// Device/Application/可视化/TlCtrl
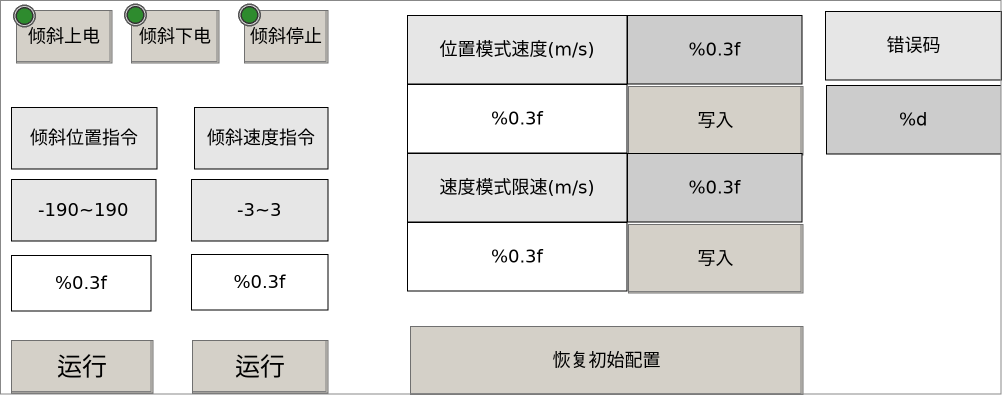
VISUALIZATION TlCtrl  // 1002x395
    Button (131,10 88x53), "倾斜下电"
        OnMouseClick: execute { GVL.Axis3Local.iMode:=0; }
    Button (16,10 96x53), "倾斜上电"
        OnMouseClick: execute { GVL.Axis3Local.iMode:=1; }
    Lamp1 (6,3 37x26), variable: GVL.Axis3Status.bServo_Enable, style: Lamp-Lamp1-Green
    Lamp1 (117,2 37x26), variable: NOT(GVL.Axis3Status.bServo_Enable), style: Lamp-Lamp1-Green
    Button (244,10 84x53), "倾斜停止"
        OnMouseClick: execute { GVL.Axis3Local.iMode:=7; }
    Lamp1 (231,2 37x26), variable: NOT(GVL.Axis3Status.Moving), style: Lamp-Lamp1-Green
    Rectangle (11,107 146x62), "倾斜位置指令"
    Rectangle (11,255 140x56), "%0.3f", text variable: TiV.rPosCmd
        OnMouseClick: write the text variable via Default, min -190, max 190
    Button (11,340 142x53), "运行"
        OnMouseClick: execute {
            GVL.Axis3Local.rPosCmd:=-GVL.TiV.rPosCmd;
            GVL.Axis3Local.iMode:=4;
            GVL.Axis3Local.bPIDEnable:=TRUE;
        }
    Rectangle (194,107 134x62), "倾斜速度指令"
    Rectangle (191,254 137x56), "%0.3f", text variable: TiV.rVelCmd
        OnMouseClick: write the text variable via Default, min -11, max 11
    Button (192,340 136x53), "运行"
        OnMouseClick: execute { GVL.Axis3Local.rVelCmd:=GVL.TiV.rVelCmd*(-1); GVL.Axis3Local.iMode:=3; }
    Rectangle (11,179 145x62), "-190~190"
    Rectangle (191,179 137x62), "-3~3"
    Rectangle (627,15 175x69), "%0.3f", text variable: Axis3Local.Pos_Vel
    Rectangle (407,15 220x69), "位置模式速度(m/s)"
    Rectangle (407,84 220x69), "%0.3f", text variable: TiV.Pos_Vel
        OnMouseClick: write the text variable via Edit, min -15.5, max 15.5
    Button (628,86 175x69), "写入"
        OnMouseClick: execute { Axis3Local.Pos_Vel:=TiV.Pos_Vel; }
    Rectangle (627,153 175x69), "%0.3f", text variable: Axis3Local.rVel_Limit
    Rectangle (407,153 220x69), "速度模式限速(m/s)"
    Rectangle (407,222 220x69), "%0.3f", text variable: TiV.rVel_Limit
        OnMouseClick: write the text variable via Edit, min -15.5, max 15.5
    Button (628,224 175x69), "写入"
        OnMouseClick: execute { Axis3Local.rVel_Limit:=TiV.rVel_Limit; }
    Button (410,326 393x69), "恢复初始配置"
        OnMouseClick: execute { Axis3Local.rVel_Limit:=3; Axis3Local.Pos_Vel:=4; }
    Rectangle (826,85 175x69), "%d", text variable: GVL.eTiErrorcode
    Rectangle (825,11 177x69), "错误码"
END_VISUALIZATION

// Device/Application/可视化/north
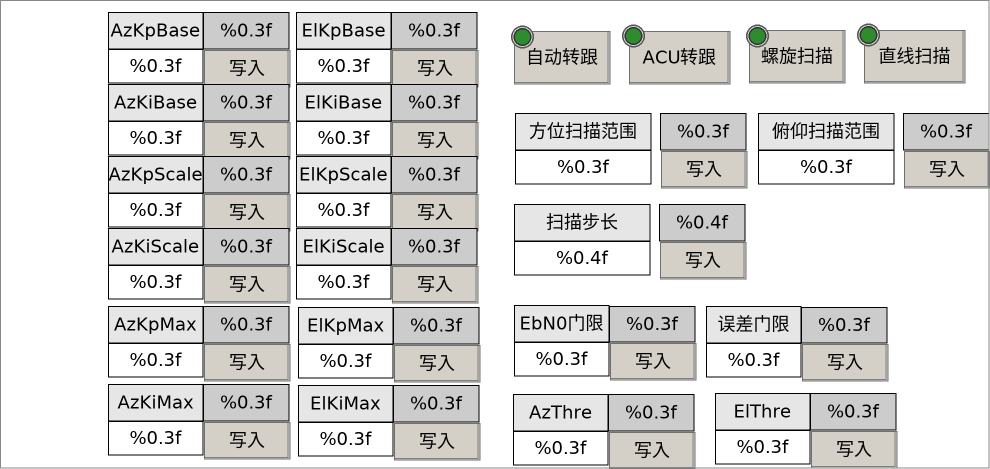
VISUALIZATION north  // 990x469
    Rectangle (203,12 86x37), "%0.3f", text variable: PersistentVars.rAzKpBase
    Rectangle (108,12 95x37), "AzKpBase"
    Rectangle (108,49 95x34), "%0.3f", text variable: GVL.rvAzKpBase
        OnMouseClick: write the text variable via Edit, min -100, max 100
    Button (204,50 86x37), "写入"
        OnMouseClick: execute { persistentvars.rAzKpBase := gvl.rvAzKpBase; }
    Rectangle (203,84 86x37), "%0.3f", text variable: PersistentVars.rAzKiBase
    Button (204,122 86x37), "写入"
        OnMouseClick: execute { persistentvars.rAzKiBase := gvl.rvAzKiBase; }
    Rectangle (203,156 86x37), "%0.3f", text variable: PersistentVars.rAzKpscale
    Button (204,194 86x37), "写入"
        OnMouseClick: execute { persistentvars.rAzKpScale := gvl.rvAzKpScale; }
    Rectangle (203,228 86x37), "%0.3f", text variable: PersistentVars.rAzKiscale
    Button (204,266 86x37), "写入"
        OnMouseClick: execute { persistentvars.rAzKiScale := gvl.rvAzKiScale; }
    Rectangle (108,84 95x37), "AzKiBase"
    Rectangle (108,121 95x34), "%0.3f", text variable: GVL.rvAzKiBase
        OnMouseClick: write the text variable via Edit, min -100, max 100
    Rectangle (108,156 95x37), "AzKpScale"
    Rectangle (108,193 95x34), "%0.3f", text variable: GVL.rvAzKpscale
        OnMouseClick: write the text variable via Edit, min -100, max 100
    Rectangle (108,228 95x37), "AzKiScale"
    Rectangle (108,265 95x34), "%0.3f", text variable: GVL.rvAzKiscale
        OnMouseClick: write the text variable via Edit, min -100, max 100
    Rectangle (391,12 86x37), "%0.3f", text variable: PersistentVars.rElKpBase
    Rectangle (296,12 95x37), "ElKpBase"
    Rectangle (296,49 95x34), "%0.3f", text variable: GVL.rvElKpBase
        OnMouseClick: write the text variable via Edit, min -100, max 100
    Button (392,50 86x37), "写入"
        OnMouseClick: execute { persistentvars.rElKpBase := gvl.rvElKpBase; }
    Rectangle (391,84 86x37), "%0.3f", text variable: PersistentVars.rElKiBase
    Button (392,122 86x37), "写入"
        OnMouseClick: execute { persistentvars.rElKiBase := gvl.rvElKiBase; }
    Rectangle (391,156 86x37), "%0.3f", text variable: PersistentVars.rElKpscale
    Button (392,194 86x37), "写入"
        OnMouseClick: execute { persistentvars.rElKpScale := gvl.rvElKpScale; }
    Rectangle (391,228 86x37), "%0.3f", text variable: PersistentVars.rElKiscale
    Button (392,266 86x37), "写入"
        OnMouseClick: execute { persistentvars.rElKiScale := gvl.rvElKiScale; }
    Rectangle (296,84 95x37), "ElKiBase"
    Rectangle (296,121 95x34), "%0.3f", text variable: GVL.rvElKiBase
        OnMouseClick: write the text variable via Edit, min -100, max 100
    Rectangle (296,156 95x37), "ElKpScale"
    Rectangle (296,193 95x34), "%0.3f", text variable: GVL.rvElKpscale
        OnMouseClick: write the text variable via Edit, min -100, max 100
    Rectangle (296,228 95x37), "ElKiScale"
    Rectangle (296,265 95x34), "%0.3f", text variable: GVL.rvElKiscale
        OnMouseClick: write the text variable via Edit, min -100, max 100
    Rectangle (203,306 86x37), "%0.3f", text variable: PersistentVars.rAzKpMax
    Rectangle (108,306 95x37), "AzKpMax"
    Rectangle (108,343 95x34), "%0.3f", text variable: GVL.rvAzKpMax
        OnMouseClick: write the text variable via Edit, min -100, max 100
    Button (204,344 86x37), "写入"
        OnMouseClick: execute { persistentvars.rAzKpMax := gvl.rvAzKpMax; }
    Rectangle (203,384 86x37), "%0.3f", text variable: PersistentVars.rAzKiMax
    Rectangle (108,384 95x37), "AzKiMax"
    Rectangle (108,421 95x34), "%0.3f", text variable: GVL.rvAzKiMax
        OnMouseClick: write the text variable via Edit, min -100, max 100
    Button (204,422 86x37), "写入"
        OnMouseClick: execute { persistentvars.rAzKiMax := gvl.rvAzKiMax; }
    Rectangle (393,307 86x37), "%0.3f", text variable: PersistentVars.rElKpMax
    Rectangle (298,307 95x37), "ElKpMax"
    Rectangle (298,344 95x34), "%0.3f", text variable: GVL.rvElKpMax
        OnMouseClick: write the text variable via Edit, min -100, max 100
    Button (394,345 86x37), "写入"
        OnMouseClick: execute { persistentvars.rElKpMax := gvl.rvElKpMax; }
    Rectangle (393,385 86x37), "%0.3f", text variable: PersistentVars.rElKiMax
    Rectangle (298,385 95x37), "ElKiMax"
    Rectangle (298,422 95x34), "%0.3f", text variable: GVL.rvElKiMax
        OnMouseClick: write the text variable via Edit, min -100, max 100
    Button (394,423 86x37), "写入"
        OnMouseClick: execute { persistentvars.rElKiMax := gvl.rvElKiMax; }
    Rectangle (608,394 86x37), "%0.3f", text variable: PersistentVars.rAzThre
    Rectangle (513,394 95x37), "AzThre"
    Rectangle (513,431 95x34), "%0.3f", text variable: GVL.rvAzThre
        OnMouseClick: write the text variable via Edit, min -100, max 100
    Button (609,432 86x37), "写入"
        OnMouseClick: execute { persistentvars.rAzThre := gvl.rvAzThre; }
    Rectangle (810,393 86x37), "%0.3f", text variable: PersistentVars.rElThre
    Rectangle (715,393 95x37), "ElThre"
    Rectangle (715,430 95x34), "%0.3f", text variable: GVL.rvElThre
        OnMouseClick: write the text variable via Edit, min -100, max 100
    Button (811,431 86x37), "写入"
        OnMouseClick: execute { persistentvars.rElThre := gvl.rvElThre; }
    Rectangle (609,306 86x36), "%0.3f", text variable: PersistentVars.rEbN0LockThre
    Rectangle (514,305 95x37), "EbN0门限"
    Rectangle (514,342 95x34), "%0.3f", text variable: GVL.rEbN0LockThreEdit
        OnMouseClick: write the text variable via Edit, min 0, max 30
    Button (610,343 86x37), "写入"
        OnMouseClick: execute { PersistentVars.rEbN0LockThre := GVL.rEbN0LockThreEdit; }
    Rectangle (660,113 86x37), "%0.3f", text variable: PersistentVars.rAzScanRange
    Rectangle (515,113 136x37), "方位扫描范围"
    Rectangle (515,150 136x34), "%0.3f", text variable: GVL.rAzScanRangeTemp
        OnMouseClick: write the text variable via Edit, min 0.1, max 1
    Button (661,151 86x37), "写入"
        OnMouseClick: execute { persistentvars.rAzScanRange := gvl.rAzScanRangeTemp; }
    Rectangle (903,113 86x37), "%0.3f", text variable: PersistentVars.rElScanRange
    Rectangle (758,113 136x37), "俯仰扫描范围"
    Rectangle (758,150 136x34), "%0.3f", text variable: GVL.rElScanRangeTemp
        OnMouseClick: write the text variable via Edit, min 0, max 1
    Button (904,151 86x37), "写入"
        OnMouseClick: execute { persistentvars.rElScanRange := gvl.rElScanRangeTemp; }
    Button (629,31 101x53), "ACU转跟"
        OnMouseClick: execute { PersistentVars.bTrackingMode:=FALSE; }
    Button (514,31 96x53), "自动转跟"
        OnMouseClick: execute { PersistentVars.bTrackingMode:=TRUE; }
    Lamp1 (504,24 37x26), variable: PersistentVars.bTrackingMode, style: Lamp-Lamp1-Green
    Lamp1 (615,23 37x26), variable: NOT(PersistentVars.bTrackingMode), style: Lamp-Lamp1-Green
    Button (864,30 101x53), "直线扫描"
        OnMouseClick: execute { PersistentVars.bSearchType:=FALSE; }
    Button (749,30 96x53), "螺旋扫描"
        OnMouseClick: execute { PersistentVars.bSearchType:=TRUE; }
    Lamp1 (739,23 37x26), variable: PersistentVars.bSearchType, style: Lamp-Lamp1-Green
    Lamp1 (850,22 37x26), variable: NOT(PersistentVars.bSearchType), style: Lamp-Lamp1-Green
    Rectangle (801,307 86x36), "%0.3f", text variable: PersistentVars.rErrorThre
    Rectangle (706,306 95x37), "误差门限"
    Rectangle (706,343 95x34), "%0.3f", text variable: GVL.rErrorTherTemp
        OnMouseClick: write the text variable via Edit, min 0, max 10
    Button (802,344 86x37), "写入"
        OnMouseClick: execute { PersistentVars.rErrorThre := GVL.rErrorTherTemp; }
    Rectangle (659,204 86x37), "%0.4f", text variable: PersistentVars.rStep
    Rectangle (514,204 136x37), "扫描步长"
    Rectangle (514,241 136x34), "%0.4f", text variable: GVL.rStepTemp
        OnMouseClick: write the text variable via Edit, min 0.0001, max 0.1
    Button (660,242 86x37), "写入"
        OnMouseClick: execute { persistentvars.rStep := gvl.rStepTemp; }
END_VISUALIZATION
